ABB RAPID module: Wizard.modx

MODULE Wizard
    PROC main()
	    ImagenesAuto;
	ENDPROC
ENDMODULE
